# EPICS autosave request: support/ebrick/2-2-3/iocBoot/iocebrick/autosave/auto_settings.req
## eBrick settings
file ebrick_settings.req P=$(P)

## User-programming settings
file userAve10_settings.req P=$(P)
file userCalcs10_settings.req P=$(P)
file userTransforms10_settings.req P=$(P)
file userStringCalcs10_settings.req P=$(P)

file sseq_settings.req P=$(P),S=Sseq1
file sseq_settings.req P=$(P),S=Sseq2
file sseq_settings.req P=$(P),S=Sseq3
